// TIA Portal project "CarroponteFB" (V16)

(* hardware
DEVICE "S7-1200 station_1"  S7-1200 Station
   slot 0: "Telaio di montaggio_0"  S7-1200 Rack  Rack  V1.0
   slot 1: "PLC_1"  CPU 1214C DC/DC/DC  6ES7 214-1AG40-0XB0  V4.1
*)

// ===== PLC "PLC_1"  CPU 1214C DC/DC/DC =====

VAR_GLOBAL   // PLC tag table "Tabella delle variabili standard"
   "START" AT %I0.0 : Bool;
   "SDown" AT %I0.1 : Bool;
   "SUp" AT %I0.2 : Bool;
   "S1" AT %I0.3 : Bool;
   "S2" AT %I0.4 : Bool;
   "S3" AT %I0.5 : Bool;
   "Left" AT %Q0.0 : Bool;
   "Right" AT %Q0.1 : Bool;
   "Down" AT %Q0.2 : Bool;
   "Up" AT %Q0.3 : Bool;
END_VAR

VAR_GLOBAL CONSTANT   // PLC tag table "Tabella delle variabili standard"
   "TEMPO_TRASCORSO" : Time := T#15s;
END_VAR

DATA_BLOCK "Carroponte_DB"   // DB1
{ S7_Optimized_Access := 'TRUE' }
VERSION : 0.1
// stored: InstanceOfName Carroponte
"Carroponte"
BEGIN
END_DATA_BLOCK

FUNCTION_BLOCK "Carroponte"   // FB1, LAD
{ S7_Optimized_Access := 'TRUE' }
VERSION : 0.1
   VAR_INPUT
      START : Bool;
      SDown : Bool;
      SUp : Bool;
      S1 : Bool;
      S2 : Bool;
      S3 : Bool;
      TEMPO_TRASCORSO : Time := T#15ms;
   END_VAR
   VAR_OUTPUT
      Left : Bool;
      Right : Bool;
      Down : Bool;
      Up : Bool;
   END_VAR
   VAR RETAIN
      HOME : Bool := true;
      Destra1 : Bool;
      Su : Bool;
      Destra2 : Bool;
      Attesa : Bool;
      Sinistra : Bool;
      Giù : Bool;
   END_VAR
   VAR
      IEC_Timer_0_Instance : TON_TIME;
   END_VAR
BEGIN

REGION Network 1
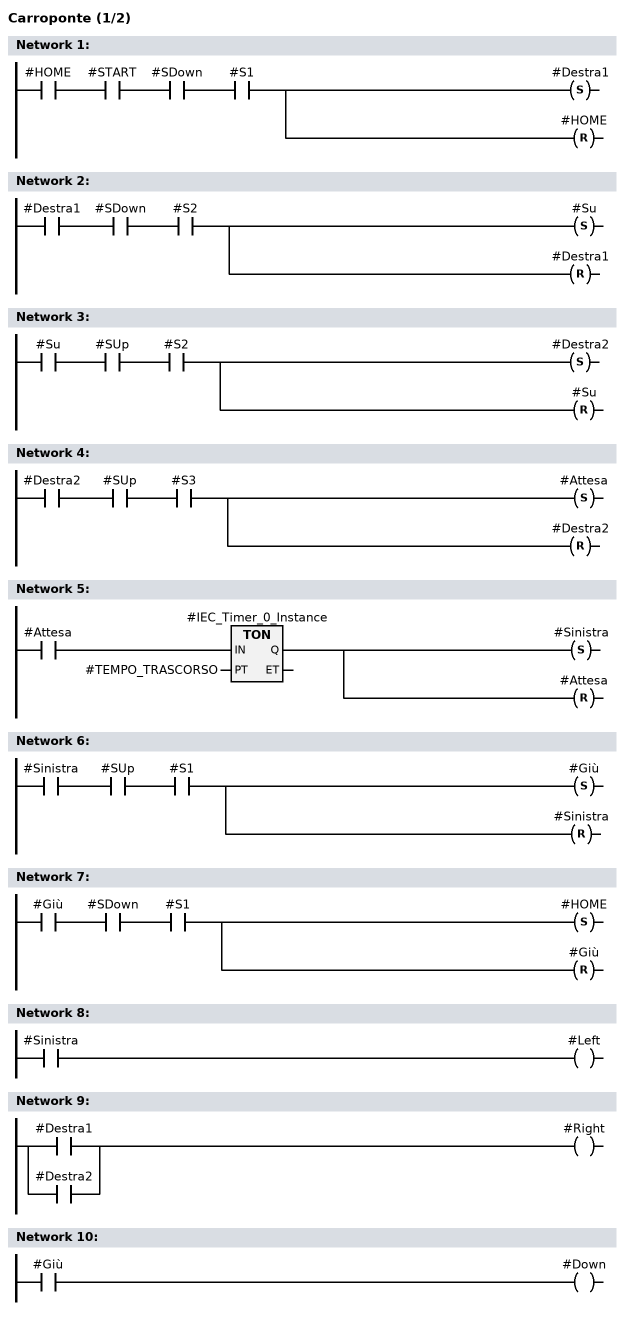
   RUNG wire#powerrail
      Contact( #HOME )
      Contact( #START )
      Contact( #SDown )
      Contact( #S1 )
      wire#w1
      S_Coil( #Destra1 )
   END_RUNG
   RUNG wire#w1
      R_Coil( #HOME )
   END_RUNG
   // the same network as SCL:
   IF #HOME AND #START AND #SDown AND #S1 THEN
       #Destra1 := TRUE;
       #HOME := FALSE;
   END_IF;
END_REGION

REGION Network 2
   RUNG wire#powerrail
      Contact( #Destra1 )
      Contact( #SDown )
      Contact( #S2 )
      wire#w1
      S_Coil( #Su )
   END_RUNG
   RUNG wire#w1
      R_Coil( #Destra1 )
   END_RUNG
   // the same network as SCL:
   IF #Destra1 AND #SDown AND #S2 THEN
       #Su := TRUE;
       #Destra1 := FALSE;
   END_IF;
END_REGION

REGION Network 3
   RUNG wire#powerrail
      Contact( #Su )
      Contact( #SUp )
      Contact( #S2 )
      wire#w1
      S_Coil( #Destra2 )
   END_RUNG
   RUNG wire#w1
      R_Coil( #Su )
   END_RUNG
   // the same network as SCL:
   IF #Su AND #SUp AND #S2 THEN
       #Destra2 := TRUE;
       #Su := FALSE;
   END_IF;
END_REGION

REGION Network 4
   RUNG wire#powerrail
      Contact( #Destra2 )
      Contact( #SUp )
      Contact( #S3 )
      wire#w1
      S_Coil( #Attesa )
   END_RUNG
   RUNG wire#w1
      R_Coil( #Destra2 )
   END_RUNG
   // the same network as SCL:
   IF #Destra2 AND #SUp AND #S3 THEN
       #Attesa := TRUE;
       #Destra2 := FALSE;
   END_IF;
END_REGION

REGION Network 5
   #IEC_Timer_0_Instance(IN := #Attesa, PT := #TEMPO_TRASCORSO);   // TON
   IF #IEC_Timer_0_Instance.Q THEN
       #Sinistra := TRUE;
       #Attesa := FALSE;
   END_IF;
END_REGION

REGION Network 6
   RUNG wire#powerrail
      Contact( #Sinistra )
      Contact( #SUp )
      Contact( #S1 )
      wire#w1
      S_Coil( #Giù )
   END_RUNG
   RUNG wire#w1
      R_Coil( #Sinistra )
   END_RUNG
   // the same network as SCL:
   IF #Sinistra AND #SUp AND #S1 THEN
       #Giù := TRUE;
       #Sinistra := FALSE;
   END_IF;
END_REGION

REGION Network 7
   RUNG wire#powerrail
      Contact( #Giù )
      Contact( #SDown )
      Contact( #S1 )
      wire#w1
      S_Coil( #HOME )
   END_RUNG
   RUNG wire#w1
      R_Coil( #Giù )
   END_RUNG
   // the same network as SCL:
   IF #Giù AND #SDown AND #S1 THEN
       #HOME := TRUE;
       #Giù := FALSE;
   END_IF;
END_REGION

REGION Network 8
   RUNG wire#powerrail
      Contact( #Sinistra )
      Coil( #Left )
   END_RUNG
   // the same network as SCL:
   #Left := #Sinistra;
END_REGION

REGION Network 9
   RUNG wire#powerrail
      Contact( #Destra1 )
      wire#w1
      Coil( #Right )
   END_RUNG
   RUNG wire#powerrail
      Contact( #Destra2 )
   END_RUNG wire#w1
   // the same network as SCL:
   #Right := #Destra1 OR #Destra2;
END_REGION

REGION Network 10
   RUNG wire#powerrail
      Contact( #Giù )
      Coil( #Down )
   END_RUNG
   // the same network as SCL:
   #Down := #Giù;
END_REGION

REGION Network 11
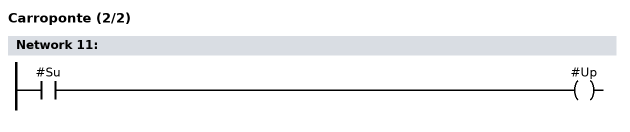
   RUNG wire#powerrail
      Contact( #Su )
      Coil( #Up )
   END_RUNG
   // the same network as SCL:
   #Up := #Su;
END_REGION
END_FUNCTION_BLOCK

ORGANIZATION_BLOCK "Main"   // OB1, LAD, ProgramCycle
TITLE = "Main Program Sweep (Cycle)"
{ S7_Optimized_Access := 'TRUE' }
VERSION : 0.1
   VAR_INPUT
      Initial_Call : Bool;   // Initial call of this OB
      Remanence : Bool;   // =True, if remanent data are available
   END_VAR
BEGIN

REGION Network 1
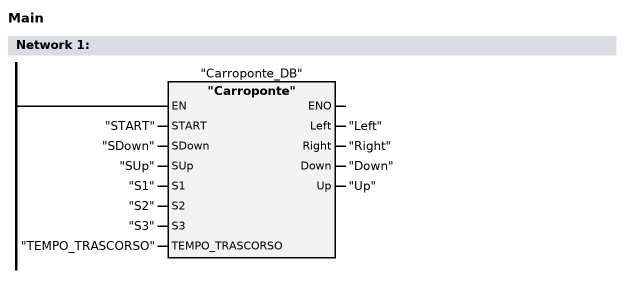
   RUNG wire#powerrail
      "Carroponte_DB"(START := "START", SDown := "SDown", SUp := "SUp", S1 := "S1", S2 := "S2", S3 := "S3", TEMPO_TRASCORSO := "TEMPO_TRASCORSO", Left => "Left", Right => "Right", Down => "Down", Up => "Up")
   END_RUNG
   // the same network as SCL:
   "Carroponte_DB"(START := "START",   // "Carroponte"
                   SDown := "SDown",
                   SUp := "SUp",
                   S1 := "S1",
                   S2 := "S2",
                   S3 := "S3",
                   TEMPO_TRASCORSO := "TEMPO_TRASCORSO",
                   Left => "Left",
                   Right => "Right",
                   Down => "Down",
                   Up => "Up");
END_REGION
END_ORGANIZATION_BLOCK